TYPE fbPistonConfig :
STRUCT
	MaxTimeToReachHome : TIME;
	MaxTimeToReachWork : TIME;
END_STRUCT
END_TYPE

(* stored: Version 1.1.0.1
   DUT fbPistonConfig: Id {4309ea9b-fad4-057d-195c-77e901d69290} *)
